PROGRAM PRG_1_PlcTask
VAR
END_VAR

PRG_LIB();
PRG_ATM();
PRG_LJ();
PRG_SPEC();
PRG_4_LOG();

END_PROGRAM

(* stored: Version 1.1.0.1, ProductVersion 3.1.4022.18
   POU PRG_1_PlcTask: Id {42048787-7ba9-4c4c-a68e-bba60d5038d8}, SpecialFunc None *)
